PROGRAM PowerMonitoring
VAR_INPUT
	comm: I_Comm;
END_VAR
VAR_OUTPUT
	phaseOK:				BOOL;
END_VAR
VAR
	Overvoltage				AT%I*: BOOL;
	Overcurrent				AT%I*: BOOL;
	VoltageGuardWarning		AT%I*: BOOL;
	VoltageGuardError		AT%I*: BOOL;
	CurrentGuardWarning		AT%I*: BOOL;
	CurrentGuardError		AT%I*: BOOL;
	Voltage					AT%I*: REAL;
	Current					AT%I*: REAL;
	ActivePower				AT%I*: REAL;
	ApparentPower			AT%I*: REAL;
	ReactivePower			AT%I*: REAL;
	PowerQualityFactor		AT%I*: REAL;
	Frequency				AT%I*: REAL;
	PowerFactor				AT%I*: REAL;
	NeutralLineCurrent		AT%I*: REAL;
	L1L2Voltage				AT%I*: REAL;
	L2L3Voltage				AT%I*: REAL;
	L3L1Voltage				AT%I*: REAL;
	MQTTTimer: 				TON := (PT:=T#10S);
	PowerWarningDelay:		TON := (PT:=T#100MS);
	PowerWarningRetain:		TOF := (PT:=T#2000MS);
	
	PowerError:				FB_EventLog;
	PowerWarning:			FB_EventLog;
	NeutralCurrentEvent:			FB_EventLog;
END_VAR

phaseOK := L1L2Voltage > 360.0 AND L2L3Voltage > 360.0 AND L3L1Voltage > 360.0;

IF NeutralLineCurrent > 0.1 THEN
	NeutralCurrentEvent.Trigger := TRUE;
	NeutralCurrentEvent.OnMessage := 	'Neutral Line Current WARNING!';
	NeutralCurrentEvent.Level := ADSLOG_MSGTYPE_WARN;
ELSIF NeutralLineCurrent > 0.3 THEN
	NeutralCurrentEvent.Trigger := TRUE;
	NeutralCurrentEvent.OnMessage := 	'Neutral Line Current ERROR!';
	NeutralCurrentEvent.Level := ADSLOG_MSGTYPE_ERROR;
ELSE
	NeutralCurrentEvent.Trigger := FALSE;
END_IF

PowerWarningDelay(IN := VoltageGuardWarning OR CurrentGuardWarning);
PowerWarningRetain(IN := PowerWarningDelay.Q);

// MQTT Section
MQTTTimer(IN:=TRUE);
IF MQTTTimer.Q OR VoltageGuardWarning OR CurrentGuardWarning THEN // publish new payload every second
	MQTTTimer(IN:=FALSE);

	comm.Publish('telescope', 'power', 'Overvoltege',	BOOL_TO_STRING(Overvoltage));
	comm.Publish('telescope', 'power', 'Overcurrent',	BOOL_TO_STRING(Overcurrent));

	comm.Publish('telescope', 'power', 'VoltageGuardWarning',	BOOL_TO_STRING(VoltageGuardWarning));
	comm.Publish('telescope', 'power', 'VoltageGuardError',		BOOL_TO_STRING(VoltageGuardError));
	comm.Publish('telescope', 'power', 'CurrentGuardWarning',	BOOL_TO_STRING(CurrentGuardWarning));
	comm.Publish('telescope', 'power', 'CurrentGuardError',		BOOL_TO_STRING(CurrentGuardError));

	comm.Publish('telescope', 'power', 'Voltage', 		REAL_TO_STRING(Voltage));
	comm.Publish('telescope', 'power', 'Current',		REAL_TO_STRING(Current));
	comm.Publish('telescope', 'power', 'ActivePower',	REAL_TO_STRING(ActivePower));
	comm.Publish('telescope', 'power', 'ApparentPower',	REAL_TO_STRING(ApparentPower));
	comm.Publish('telescope', 'power', 'ReactivePower',	REAL_TO_STRING(ReactivePower));
	comm.Publish('telescope', 'power', 'PowerQualityFactor',	REAL_TO_STRING(PowerQualityFactor));
	comm.Publish('telescope', 'power', 'Frequency',		REAL_TO_STRING(Frequency));
	comm.Publish('telescope', 'power', 'PowerFactor',	REAL_TO_STRING(PowerFactor));
	comm.Publish('telescope', 'power', 'NeutralLineCurrent',	REAL_TO_STRING(NeutralLineCurrent));

	comm.Publish('telescope', 'power', 'L1L2Voltage',	REAL_TO_STRING(L1L2Voltage));
	comm.Publish('telescope', 'power', 'L2L3Voltage',	REAL_TO_STRING(L2L3Voltage));
	comm.Publish('telescope', 'power', 'L3L1Voltage',	REAL_TO_STRING(L3L1Voltage));	
END_IF

// EventLog section
PowerError(	
	Trigger := 		VoltageGuardError OR CurrentGuardError, 
	Level := 		ADSLOG_MSGTYPE_ERROR,
	FormatString :=	'%s',
	OnMessage := 	'electrical power:	ERROR!');
	
PowerWarning(	
	Trigger := 		PowerWarningRetain.Q, 
	Level := 		ADSLOG_MSGTYPE_WARN,
	FormatString :=	'%s',
	OnMessage := 	'electrical power:	WARNING!');

NeutralCurrentEvent(
	FormatString :=	'%s',
	OnMessage := 	'electrical power:	WARNING!');

END_PROGRAM

(* stored: Version 1.1.0.1, ProductVersion 3.1.4026.8
   POU PowerMonitoring: Id {8c6b81b0-5d31-4dfd-9f1e-620164ef7757}, SpecialFunc None *)
